FUNCTION_BLOCK FB_RCC_Valves
VAR_INPUT
      RCC_VRC_01 : FB_VRC_NC_ClsLS;
      RCC_VRC_02 : FB_VRC;
      RCC_VRC_03 : FB_VRC_NC_ClsLS;
      RCC_VRC_04 : FB_VRC_NC_ClsLS;

      RCC_GCP_01 : FB_901_ECAT;
      RCC_GCP_01_INTERLOCK_SETPOINT : REAL;
END_VAR
VAR
    RCC_VRC_01_OPEN_OK : BOOL;
    RCC_VRC_02_OPEN_OK : BOOL;
    RCC_VRC_03_OPEN_OK : BOOL;
    RCC_VRC_04_OPEN_OK : BOOL;
END_VAR

RCC_GCP_01(PG=>);

(* Valve can open only when RCC-VRC-02 and 03 are closed*)
RCC_VRC_01_OPEN_OK := ( RCC_VRC_02.iq_stValve.i_xClsLS AND NOT RCC_VRC_02.iq_stValve.q_xOPN_DO ) AND
                                    ( RCC_VRC_03.iq_stValve.i_xClsLS AND NOT RCC_VRC_03.iq_stValve.q_xOPN_DO ) ;

RCC_VRC_01(i_xExtILK_OK := RCC_VRC_01_OPEN_OK,
                i_xOverrideMode := xSystemOverrideMode_RCC,
                 iq_stValve=> );

(* Valve can open only when RCC-VRC-01 and 04 are closed*)
RCC_VRC_02_OPEN_OK := ( RCC_VRC_01.iq_stValve.i_xClsLS AND NOT RCC_VRC_01.iq_stValve.q_xOPN_DO ) AND
                                    ( RCC_VRC_04.iq_stValve.i_xClsLS AND NOT RCC_VRC_04.iq_stValve.q_xOPN_DO );

RCC_VRC_02(i_xExtILK_OK := RCC_VRC_02_OPEN_OK,
                i_xOverrideMode := xSystemOverrideMode_RCC,
                 iq_stValve=> );

(* Valve can open only when RCC-GCP-01 reading < setpoint Torr and RCC-VRC-01 and 04 are closed*)
RCC_VRC_03_OPEN_OK := (RCC_GCP_01.PG.rPRESS < RCC_GCP_01_INTERLOCK_SETPOINT and RCC_GCP_01.PG.xPRESS_OK ) AND
                                 ( RCC_VRC_01.iq_stValve.i_xClsLS AND NOT RCC_VRC_01.iq_stValve.q_xOPN_DO ) AND
                                              ( RCC_VRC_04.iq_stValve.i_xClsLS AND NOT RCC_VRC_04.iq_stValve.q_xOPN_DO );

RCC_VRC_03(i_xExtILK_OK := RCC_VRC_03_OPEN_OK,
                i_xOverrideMode := xSystemOverrideMode_RCC,
                 iq_stValve=> );

(* Valve can open only when RCC-VRC-02 and 03 are closed*)
RCC_VRC_04_OPEN_OK := ( RCC_VRC_02.iq_stValve.i_xClsLS AND NOT RCC_VRC_02.iq_stValve.q_xOPN_DO ) AND
                                      ( RCC_VRC_03.iq_stValve.i_xClsLS AND NOT RCC_VRC_03.iq_stValve.q_xOPN_DO ) ;

RCC_VRC_04(i_xExtILK_OK := RCC_VRC_04_OPEN_OK,
                i_xOverrideMode := xSystemOverrideMode_RCC,
                 iq_stValve=> );

END_FUNCTION_BLOCK

(* stored: Version 1.1.0.1, ProductVersion 3.1.4024.12
   POU FB_RCC_Valves: Id {aeda5aca-2ac4-452c-9a2a-9422247ebe85}, SpecialFunc None *)
